PROGRAM MAIN
VAR
	udp1 : UdpReceiver;
END_VAR

udp1();

END_PROGRAM

(* stored: Version 1.1.0.1, ProductVersion 3.1.0.34
   POU MAIN: Id {f9351a7e-7ff5-47bf-9b6f-657a6a76e82c}, SpecialFunc None *)
